# EPICS autosave request: iocBoot/iocCygwin/auto_positions.req
$(P)m1.OFF
$(P)m1.DVAL
$(P)m2.OFF
$(P)m2.DVAL
$(P)m3.OFF
$(P)m3.DVAL
$(P)m4.OFF
$(P)m4.DVAL
$(P)m5.OFF
$(P)m5.DVAL
$(P)m6.OFF
$(P)m6.DVAL
$(P)m7.OFF
$(P)m7.DVAL
$(P)m8.OFF
$(P)m8.DVAL
